Staubli VAL3: uniqueNum.pgx

public program uniqueNum(num& x_nInput[], num& x_nResult[])
  local num l_nCoutner
  local num l_nElement
  local num l_nLength
  local string l_sString
  local num l_nBuffer
begin

//  l_nLength = size(x_sInput)
//  l_nCoutner = 0
//  resize(x_sResult,1,1)
//  resize(sStringBuffer,1,1)

//  for l_nElement = 0 to l_nLength-1

//    if l_nElement = 0
//      append(x_sResult)
//      x_sResult[size(x_sResult)-1] = x_nInput[l_nElement]
//    else

//      for l_nBuffer = 0 to size(x_sResult)-1
//        if x_sInput[l_nElement] != x_sResult[l_nBuffer]
//          append(x_sResult)
//          x_sResult[size(x_sResult)-1] = x_nInput[l_nElement]
//        endIf

//      endFor

//    endIf

//  endFor

//  delete(x_sResult[0])

end
